{attribute addProperty BoxType "EL3202-0030-0022"}
{attribute addProperty Id "RTD_Inputs_ChannelAT %I*ARRAY[0..2] OF RTD_Inputs_Channel_B51B79FC16220.250WcStateAT %I*WcState_98A4DF7520.250InfoDataAT %I*InfoData_BC63D37F80100"}
{attribute addProperty CRC "1730284832"}
{attribute addProperty SizeInBites "244"}
{attribute addProperty SizeInBytes "30.5"}
TYPE EL3202_CEE8F25A :
STRUCT
	{attribute addProperty Name "RTD_Inputs_Channel"}
	RTD_Inputs_Channel : ARRAY[0..2] OF RTD_Inputs_Channel_B51B79FC;
	{attribute addProperty Name "WcState"}
	WcState : WcState_98A4DF75;
	{attribute addProperty Name "InfoData"}
	InfoData : InfoData_BC63D37F;
END_STRUCT
END_TYPE

(* stored: Version 1.2.0.0, ProductVersion 3.1.4024.9
   DUT EL3202_CEE8F25A: Id {5d305ef3-9853-4a1d-937d-e14b74a185d7} *)
